FUNCTION_BLOCK FINAL FB_TimeManagement
VAR_IN_OUT
	Control				: ST_System;
	Control_SP			: ST_System_SP;
END_VAR
VAR
	_fb_CurrentTicks	: GETCPUCOUNTER;
	_fb_LocalSystemTime	: FB_LocalSystemTime;
	_CurrentScan		: DWORD := 0;
	_LastScan			: DWORD := 0;
	_LastScanTime		: DWORD := 0;
	_Timer_ET			: DINT;
	_Firstscan			: R_TRIG;
	_MinutePulse		: R_TRIG;
	_HourPulse			: R_TRIG;
	_fb_GetThisTaskIdx	: GETCURTASKINDEX;
	_TaskIndex			: BYTE;
	_TaskCycleCount		: UDINT;
	_TaskCycleCountLast	: UDINT;
	_TaskStarting		: BOOL;
	_StrobeTimer		: TON;
END_VAR
VAR CONSTANT
	_ticksInSecond		: DINT := 10000000;
END_VAR

A_FirstCycle();
A_LastScanTime();
A_Strobes();
A_SyncSystemTime();
A_TimePulses();
A_UpTime();

ACTION A_FirstCycle:
_fb_GetThisTaskIdx(INDEX => _TaskIndex);
_TaskCycleCount := _TaskInfo[BYTE_TO_INT(_TaskIndex)].CycleCount;

IF _TaskCycleCount > (_TaskCycleCountLast+100) THEN
	_TaskStarting := 1;
ELSE
	_TaskStarting := 0;	
END_IF
_TaskCycleCountLast := _TaskCycleCount;

_firstscan(CLK:=_TaskStarting);

IF _firstscan.Q THEN
	Control.SystemTime.FirstCycle := TRUE;
ELSE
	Control.SystemTime.FirstCycle := FALSE;
END_IF
END_ACTION

ACTION A_LastScanTime:
_fb_CurrentTicks();
_currentScan := _fb_CurrentTicks.cpuCntLoDW;

IF _lastScan > 0 THEN
	_lastScanTime := _currentScan - _lastScan;
	//Convert to seconds
	Control.SystemTime.ScanTime := DWORD_TO_REAL(_lastScanTime) / DINT_TO_REAL(_ticksInSecond);
END_IF

_lastScan := _currentScan;
END_ACTION

ACTION A_Strobes:
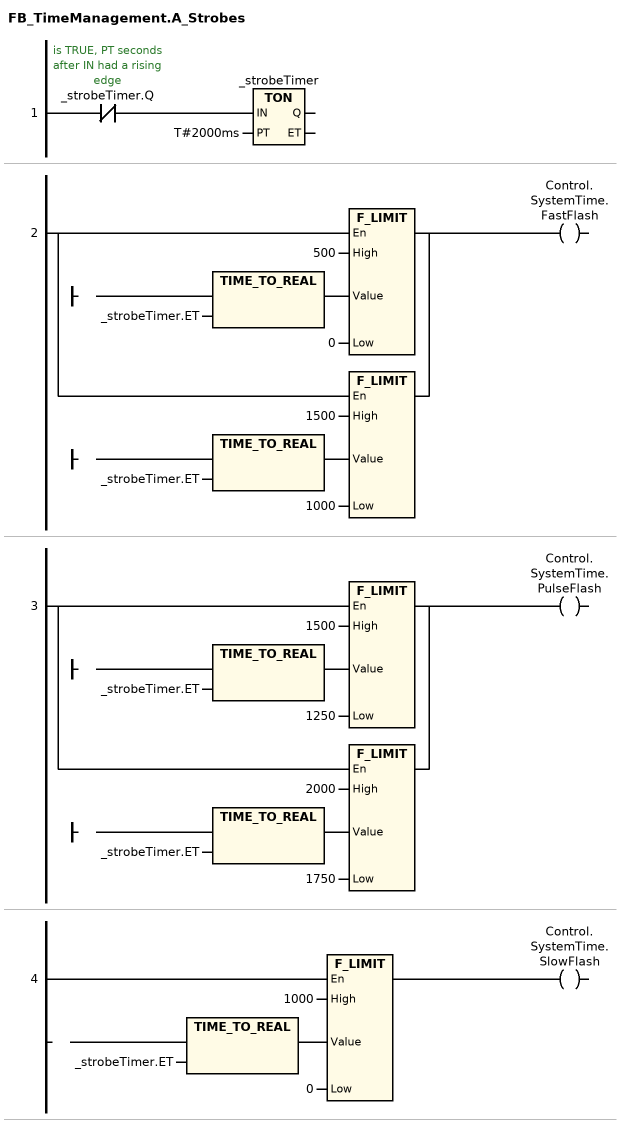
// NETWORK 1
//   _strobeTimer.Q: is TRUE, PT seconds after IN had a rising edge
_strobeTimer(IN := NOT _strobeTimer.Q, PT := T#2000ms); // TON

// NETWORK 2
//   _strobeTimer.ET: elapsed time
Control.SystemTime.FastFlash := F_LIMIT(En := TRUE, High := 500, Value := TIME_TO_REAL(_strobeTimer.ET), Low := 0) OR F_LIMIT(En := TRUE, High := 1500, Value := TIME_TO_REAL(_strobeTimer.ET), Low := 1000);

// NETWORK 3
//   _strobeTimer.ET: elapsed time
Control.SystemTime.PulseFlash := F_LIMIT(En := TRUE, High := 1500, Value := TIME_TO_REAL(_strobeTimer.ET), Low := 1250) OR F_LIMIT(En := TRUE, High := 2000, Value := TIME_TO_REAL(_strobeTimer.ET), Low := 1750);

// NETWORK 4
//   _strobeTimer.ET: elapsed time
Control.SystemTime.SlowFlash := F_LIMIT(En := TRUE, High := 1000, Value := TIME_TO_REAL(_strobeTimer.ET), Low := 0);
END_ACTION

ACTION A_SyncSystemTime:
_fb_LocalSystemTime(sNetID := '', bEnable := TRUE, dwCycle := 15, dwOpt := 1, tTimeout := DEFAULT_ADS_TIMEOUT);
IF _fb_LocalSystemTime.bValid THEN
	Control.SystemTime.CurrentTime := _fb_LocalSystemTime.systemTime;
END_IF
END_ACTION

ACTION A_TimePulses:
//Second Pulse
_timer_ET := _timer_ET + DWORD_TO_DINT(_lastScanTime);
IF _timer_ET >= _ticksInSecond THEN 
	Control.SystemTime.SecondPulse := TRUE;
	Control.SystemTime.SecondsNow := TO_DWORD(SYSTEMTIME_TO_DT(Control.SystemTime.CurrentTime));
	_timer_ET := 0;
ELSE
	Control.SystemTime.SecondPulse := FALSE;
END_IF

//Minute Pulse
_MinutePulse(CLK := Control.SystemTime.CurrentTime.wSecond = 0);
Control.SystemTime.MinutePulse :=  _MinutePulse.Q;

//Hour Pulse
_HourPulse(CLK := Control.SystemTime.CurrentTime.wMinute = 0);
Control.SystemTime.HourPulse :=  _HourPulse.Q;

//Midnight Pulse
IF WORD_TO_INT(Control.SystemTime.CurrentTime.wDay) <> Control_SP.TimeManagement.PreviousDay THEN
	Control.SystemTime.MidnightPulse := TRUE;
	Control_SP.TimeManagement.PreviousDay := WORD_TO_INT(Control.SystemTime.CurrentTime.wDay);
ELSE
	Control.SystemTime.MidnightPulse := FALSE;
END_IF
END_ACTION

ACTION A_UpTime:
IF Control.SystemTime.SecondPulse THEN
	//Up time since last reset
	Control.SystemTime.UpTime.Seconds := Control.SystemTime.UpTime.Seconds + 1;
	IF Control.SystemTime.UpTime.Seconds >= 60 THEN 
		Control.SystemTime.UpTime.Minutes := Control.SystemTime.UpTime.Minutes + 1;
		Control.SystemTime.UpTime.Seconds := 0;
	END_IF
	IF Control.SystemTime.UpTime.Minutes >= 60 THEN 
		Control.SystemTime.UpTime.Hours := Control.SystemTime.UpTime.Hours + 1;
		Control.SystemTime.UpTime.Minutes := 0;
	END_IF
	IF Control.SystemTime.UpTime.Hours >= 24 THEN 
		Control.SystemTime.UpTime.Days := Control.SystemTime.UpTime.Days + 1;
		Control.SystemTime.UpTime.Hours := 0;
	END_IF
	
	//Total up time
	Control_SP.TimeManagement.TotalUpTime.Seconds := Control_SP.TimeManagement.TotalUpTime.Seconds + 1;
	IF Control_SP.TimeManagement.TotalUpTime.Seconds >= 60 THEN 
		Control_SP.TimeManagement.TotalUpTime.Minutes := Control_SP.TimeManagement.TotalUpTime.Minutes + 1;
		Control_SP.TimeManagement.TotalUpTime.Seconds := 0;
	END_IF
	IF Control_SP.TimeManagement.TotalUpTime.Minutes >= 60 THEN 
		Control_SP.TimeManagement.TotalUpTime.Hours := Control_SP.TimeManagement.TotalUpTime.Hours + 1;
		Control_SP.TimeManagement.TotalUpTime.Minutes := 0;
	END_IF
	IF Control_SP.TimeManagement.TotalUpTime.Hours >= 24 THEN 
		Control_SP.TimeManagement.TotalUpTime.Days := Control_SP.TimeManagement.TotalUpTime.Days + 1;
		Control_SP.TimeManagement.TotalUpTime.Hours := 0;
	END_IF
END_IF
END_ACTION

END_FUNCTION_BLOCK

(* stored: Version 1.1.0.1, ProductVersion 3.1.4024.3
   POU FB_TimeManagement: Id {975fdb8f-7a89-4b70-8ffc-4e4ed2f51fc3}, SpecialFunc None
   Action A_FirstCycle: Id {3a460d9d-cf24-44c7-90fa-34a938acc8b2}
   Action A_LastScanTime: Id {a33d16e1-b93a-43c0-8d4b-8073d24ffe0d}
   Action A_Strobes: Id {a9c867b5-2c54-4418-98ee-bbbf290fe418}
   Action A_SyncSystemTime: Id {e7263b84-2d59-4eb2-af20-779c52a5518b}
   Action A_TimePulses: Id {d3adb398-20dc-4798-8f4a-889bb17c9470}
   Action A_UpTime: Id {3c8d1c80-a152-4c57-8088-34dc86e1e8e3} *)
